(* CoDeSys 2.3.9.11 project: Slunce_vypocet_pohybu_po_obloze_SUNSET.pro *)
(* Libraries: Building_common.lib 26.8.08 09:44:31, SysLibTime.lib 5.10.04 10:39:34, D:\_WAGO\IO_Pro_CAA\library\DaylightSaving.lib 22.2.07 11:46:44, SysLibRtc.lib 5.10.04 10:37:42, D:\_WAGO\IO_Pro_CAA\library\WagoLibDaylightSaving.lib 19.9.06 14:57:10, Standard.lib 22.11.04 11:21:12, SYSLIBCALLBACK.LIB 20.4.05 11:04:48 *)

(* PLC configuration (modules and I/O channels)
K-Bus [K_Bus] node 0, in %IB0 out %QB0
Fieldbus variables [FB_VARS] node 1, in %IB0 out %QB0
*)

(* Task configuration *)
TASK slunce (PRIORITY := 15, INTERVAL := T#1000ms);
	Vypocet_pohybu_slunce();
END_TASK

(* POU Vypocet_pohybu_slunce, CFC *)
PROGRAM Vypocet_pohybu_slunce
(*Program vypocte pohyb slunce po obloze na zaklade aktualnicho data a casu v systemu,
Zemepisna sirka/delka jsou nastavena na Prahu, lze libovolne zmenit.
Vystupnimi hodnotami jsou Azimut a Elevace. Pokud je Elevace<0 - Slunce zapadlo.
Vytvoreno pro procesory s 32 bitovou architekturou.
Program se spousti kazdou 1 s, jako cyklický task.
Testovano na 750-841, 750-873 	
2009-07-13 Ondrej Dolejs*)

VAR
	Pohyb_slunce: Fb_Sunset;
	AktualniCas: DT;
	UTCiCas: DT;		(*Odpovídá casu GMT, rozdíl pouze v rozsahu [s]*)
	ZemepisnaSirka: 	REAL := 50.083333333;		(*Praha 50 stupnu a 5 minut N, prepocteno stupne + minuty/60*)
	ZemepisnaDelka: REAL := 14.433333333;		(*Praha 14 stupnu a 26 minut E, prepocteno stupne + minuty/60*)
	Elevace: REAL;		(*uhel slunce nad obzorem*)
	Azimut: REAL;			(*Sever 0 stupnu, jih 180 stupnu*)
	leto: BOOL;			(*TRUE, když je leto*)
	DenVtydnu: BYTE;		(*Pondeli=1, utery=2,...., nedele=7*)
END_VAR
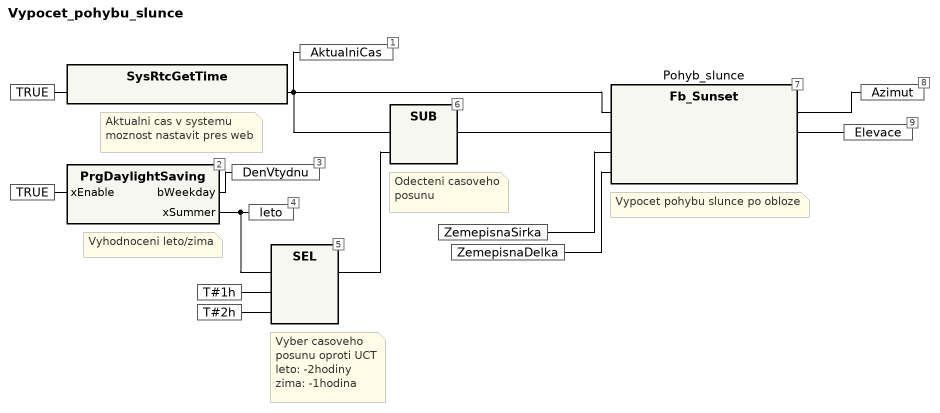
_CFC_ (* Continuous Function Chart, elements in execution order *)
#0 SysRtcGetTime(TRUE)
(* Vyber casoveho / posunu oproti UCT / leto: -2hodiny / zima: -1hodina *)
(* Aktualni cas v systemu / moznost nastavit pres web *)
(* Odecteni casoveho / posunu *)
(* Vypocet pohybu slunce po obloze *)
#1 AktualniCas <= #0
#2 PrgDaylightSaving(xEnable: TRUE)
#3 DenVtydnu <= #2.bWeekday
#4 leto <= #2.xSummer
#5 SEL(#2.xSummer, T#1h, T#2h)
#6 SUB(#0, #5)
#7 Pohyb_slunce:Fb_Sunset(#0, #6, ZemepisnaSirka, ZemepisnaDelka)
#8 Azimut <= #7.out 1
#9 Elevace <= #7.out 2
(* Vyhodnoceni leto/zima *)
_END_CFC_
END_PROGRAM
